{attribute 'linkalways'} 
{attribute 'no_explicit_call' := 'This FB is a CLASS and must be accessed using methods or properties'}
{attribute 'enable_dynamic_creation'}
FUNCTION_BLOCK Node_RGBA_CYAN EXTENDS VisionNode
VAR
    out : _TcVnVector4_LREAL;
END_VAR

METHOD PUBLIC  Clone : I_Node
VAR
	pNode : POINTER TO Node_RGBA_CYAN;
END_VAR
pNode := __NEW(Node_RGBA_CYAN);
Clone := pNode^;
END_METHOD

METHOD FB_init : BOOL
VAR_INPUT
	bInitRetains : BOOL; // if TRUE, the retain variables are initialized (warm start / cold start)
	bInCopyCode : BOOL;  // if TRUE, the instance afterwards gets moved into the copy code (online change)
END_VAR
AddOutput('out', out);
END_METHOD

METHOD PROTECTED OnExecute : HRESULT
out.Value := GVL_COLOURS.RGBA_CYAN;
END_METHOD

METHOD PUBLIC PreExecutionCheck
VAR_INPUT
	Check : I_PreExecutionChecks;
END_VAR
END_METHOD

END_FUNCTION_BLOCK

(* stored: Version 1.1.0.1, ProductVersion 3.1.4024.13
   POU Node_RGBA_CYAN: Id {34ed5850-3422-036c-17d5-3fa0113d3b59}, SpecialFunc None
   Folder Constructor: Id {8d22d9c5-a43e-06e3-1c14-af1c703fdf0d}
   Method Clone: Id {69edb072-a18a-0493-2715-4077b7bae86a}
   Method FB_init: Id {9c3b318c-ad03-07bb-3b7c-a97a19e6995f}
   Method OnExecute: Id {c952d356-bca9-0718-3aeb-78899ccba406}
   Method PreExecutionCheck: Id {e8f9f793-90fd-0ad8-2a11-bde31f0f796e} *)
